Staubli VAL3: refreshDynamic.pgx

program refreshDynamic()
begin
  // DO NOT CHANGE
  nRefresh=clock()
  use:bUseRefresh=false
  //
  // ADD HERE
  //
  // build the list
  call buildList()
  call use:listempty()
  call use:listadd(sList)
  //
  //
  // refresh the cursor
  use:nView=nView
  // refresh the list
  call use:listupdate(0)
end
